// TIA Portal V17 export
// export: Created 2023-04-03T06:31:29.5539374Z, ExportSetting WithDefaults, DisplayName Totally Integrated Automation Portal, DisplayVersion V17 Update 4, DisplayName TIA Portal Openness, DisplayVersion V17 Update 4, DisplayName TIA Portal Version Control Interface, DisplayVersion V17, DisplayName STEP 7 Professional, DisplayVersion V17 Update 4, DisplayName STEP 7 Safety, DisplayVersion V17, DisplayName WinCC Professional, DisplayVersion V17 Update 4
DATA_BLOCK "PN"   // DB11
{ S7_Optimized_Access := 'TRUE' }
VERSION : 0.1
// stored: AutoNumber false, DBAccessibleFromOPCUA true, DBAccessibleFromWebserver true, IsOnlyStoredInLoadMemory false, IsRetainMemResEnabled false, IsWriteProtectedInAS false, MemoryReserve 100
   VAR
      DevOk : Array[0..1023] of Bool;
      FltDev : Array[0..1023] of Bool;
      R : "PN Read";
      W { S7_SetPoint := 'True'} : "PN Write";
      RV_R { S7_SetPoint := 'True'} : Int;
      RV_W { S7_SetPoint := 'True'} : Int;
      xStopCmd : Bool;
      xStandByCmd : Bool;
      xRunCmd : Bool;
      xFltCmd : Bool;
      xFltClearCmd : Bool;
      iKeepAlive : Int;
      SS1 : Struct
         rPacRef : Real;
         rQacRef : Real;
      END_STRUCT;
      SS2 : Struct
         rPacRef : Real;
         rQacRef : Real;
      END_STRUCT;
      MVSKID : Struct
         xCircBrkCloseCmd : Bool;
         xCircBrkOpenCmd : Bool;
      END_STRUCT;
   END_VAR
BEGIN
END_DATA_BLOCK
